{attribute 'GeneratedUsingTerminal: EJ6224-0000-0016'}
{attribute addProperty BoxType "EJ6224-0000-0016"}
{attribute addProperty Id "Device_DiagAT %I*BOOL1Device_StateAT %I*BOOL1"}
{attribute addProperty CRC "2703295896"}
{attribute addProperty Size "2"}
TYPE DeviceState_Inputs_Device_A1210598 :
STRUCT
	{attribute addProperty Name "Device_Diag"}
	Device_Diag AT %I* : BOOL;
	{attribute addProperty Name "Device_State"}
	Device_State AT %I* : BOOL;
END_STRUCT
END_TYPE

(* stored: Version 1.2.0.0, ProductVersion 3.1.4024.9
   DUT DeviceState_Inputs_Device_A1210598: Id {f4518826-aae0-4a40-bbe9-a6c095d0c363} *)
